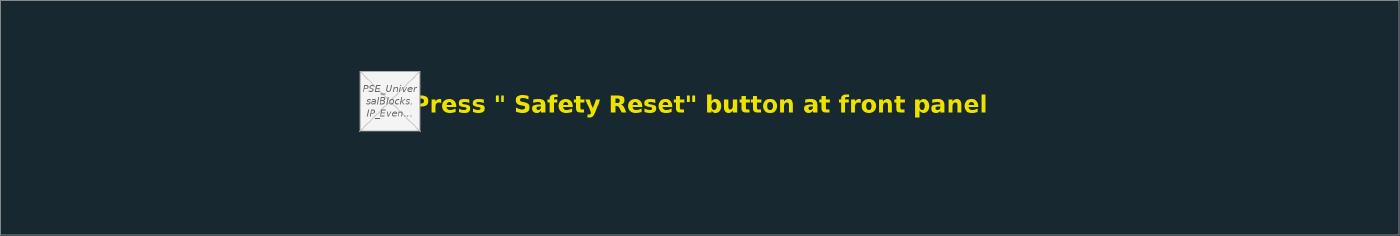
VISUALIZATION InitializingStartSafetySystem  // 1480x250
    Label (0,95 1480x30), "Press " Safety Reset" button at front panel"
    Image (380,75 64x64), image: PSE_UniversalBlocks.IP_EventSeverity.info
END_VISUALIZATION

(* stored: Version 1.1.0.1, ProductVersion 3.1.4024.9
   Visu InitializingStartSafetySystem: Id {d1ce2e60-e650-435e-aa7d-ccb4651b9484} *)
